{attribute 'GeneratedUsingTerminal: EP9224-1037-0017'}
{attribute addProperty BoxType "EP9224-1037-0017"}
{attribute addProperty Id "EtcSlaveTerminalBaseInfoDataAT %I*InfoData_6F19DB2B2"}
{attribute addProperty CRC "2874840167"}
{attribute addProperty Size "2"}
TYPE EP9224_AB5A9467 EXTENDS EtcSlaveTerminalBase :
STRUCT
	{attribute addProperty Name "InfoData"}
	InfoData : InfoData_6F19DB2B;
END_STRUCT
END_TYPE

(* stored: Version 1.2.0.0, ProductVersion 3.1.4024.9
   DUT EP9224_AB5A9467: Id {d10a54f4-c95b-4903-8395-581b400c176a} *)
